// TIA Portal project "tia_portal_to_pyhton_V18_1" (V18)

(* hardware
DEVICE "S7-1200 station_4"  S7-1200 Station
   slot 0: "Rack_0"  S7-1200 Rack  Rack  V1.0
   slot 1: "PLC_4"  CPU 1212C AC/DC/Rly  6ES7 212-1BE40-0XB0  V4.1
*)

// ===== PLC "PLC_4"  CPU 1212C AC/DC/Rly =====

VAR_GLOBAL   // PLC tag table "Default tag table"
   "Tag_2" AT %I0.0 : Bool;
   "Tag_3" AT %I0.3 : Bool;
END_VAR

VAR_GLOBAL   // PLC tag table "Tag table_1"
   "Kapı_Açık" AT %Q0.0 : Bool;   // Kapı_Açık
   "Tag_1" AT %MD10 : DWord;
   "Kapı_Kapalı" AT %Q0.1 : Bool;
   "Buzzer" AT %Q0.2 : Bool;
END_VAR

DATA_BLOCK "Data_block_1"   // DB1
{ S7_Optimized_Access := 'FALSE' }
VERSION : 0.1
   VAR
      total_prod : Int := 400;
      prod_rate : Real := 4.6;
      Message : String := 'Baret';
   END_VAR
BEGIN
END_DATA_BLOCK

// folder: System blocks/Program resources

DATA_BLOCK "TON_1"   // DB3
{ S7_Optimized_Access := 'TRUE' }
AUTHOR : Simatic
FAMILY : IEC
NAME : IEC_TMR
VERSION : 1.0
// stored: InstanceOfName IEC_TIMER
"IEC_TIMER"
BEGIN
END_DATA_BLOCK

// folder: (top level)

FUNCTION "Block_1" : Void   // FC1, LAD
{ S7_Optimized_Access := 'FALSE' }
VERSION : 0.1
BEGIN

REGION Network 1: PLC DEĞER TAŞIMA
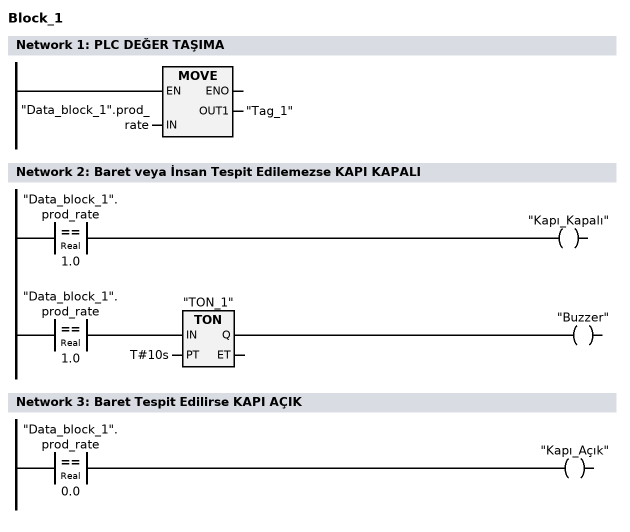
   RUNG wire#powerrail
      Move(in := "Data_block_1".prod_rate, out1 => "Tag_1")
   END_RUNG
   // the same network as SCL:
   "Tag_1" := "Data_block_1".prod_rate;
END_REGION

REGION Network 2: Baret veya İnsan Tespit Edilemezse KAPI KAPALI
   "Kapı_Kapalı" := "Data_block_1".prod_rate = 1.0;
   "TON_1".TON(IN := "Data_block_1".prod_rate = 1.0, PT := T#10s);
   "Buzzer" := "TON_1".Q;
END_REGION

REGION Network 3: Baret Tespit Edilirse KAPI AÇIK
   RUNG wire#powerrail
      { S7_Templates := "SrcType := Real" } EQ_Contact(in1 := "Data_block_1".prod_rate, in2 := 0.0)
      Coil( "Kapı_Açık" )
   END_RUNG
   // the same network as SCL:
   "Kapı_Açık" := "Data_block_1".prod_rate = 0.0;
END_REGION
END_FUNCTION

ORGANIZATION_BLOCK "Main"   // OB1, LAD, ProgramCycle
TITLE = "Main Program Sweep (Cycle)"
{ S7_Optimized_Access := 'TRUE' }
VERSION : 0.1
   VAR_INPUT
      Initial_Call : Bool;   // Initial call of this OB
      Remanence : Bool;   // =True, if remanent data are available
   END_VAR
BEGIN

REGION Network 1
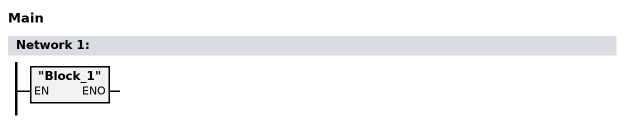
   RUNG wire#powerrail
      "Block_1"()
   END_RUNG
   // the same network as SCL:
   "Block_1"();
END_REGION
END_ORGANIZATION_BLOCK